Universal Robots PolyScope program: fill_sugar.urp

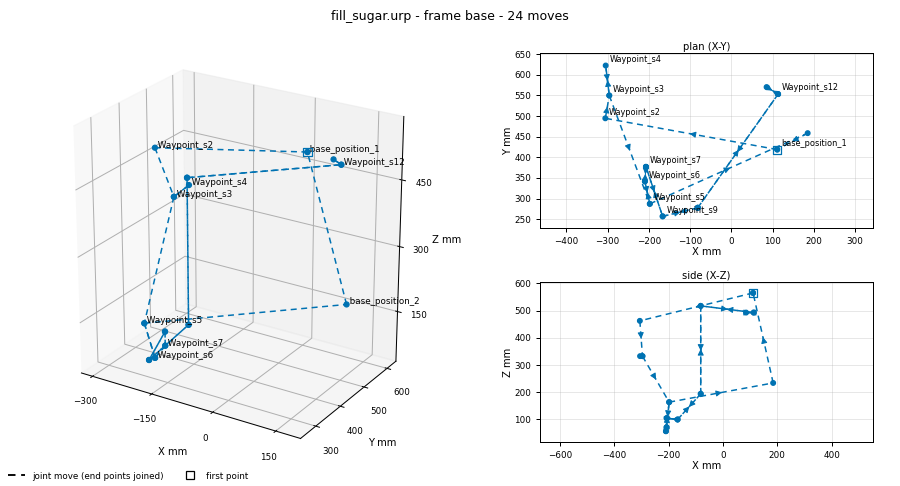
[picture p0: tool path of fill_sugar.urp in frame base, 24 of 24 moves have a stored position in this frame; points joined in program order, loops and branches not executed]
Program fill_sugar (installation=default directory=/programs/Nicolas_Arteaga createdIn=5.12.4.1101661 lastSavedIn=5.12.4.1101661 robotSerialNumber=20225502378)
Calibrated DH parameters: a=[0.00022, -0.425328, -0.389701, 0.000059, 0.000065, 0]; d=[0.162608, 0.803456, 9.992211, -10.662202, 0.099702, 0.099559]; alpha=[1.570756, 0.001543, 0.004316, 1.570651, -1.570122, 0]; deltaTheta=[0, 0.002917, 0.116094, -0.119008, 0, -0.000001]
Robot Program (runOnlyOnce=true)
  'The Sugar Workflow opens the funnel with the sugar the time needed for the amount, moves the spoon into the center of the machine and comes back'
  MoveJ speed 60 deg/s, acceleration 80 deg/s^2 (useActiveTCP=true) feature=Base
    'Use either the register for CPEE or a local parameter like 0.5'
    sugar_amount := GP_int_in[0]
    SuppressedNode
      sugar_amount := 1.5
    Waypoint base_position_1: TCP in base x=110.873 y=418.875 z=565.206 mm, rx=-1.5602 ry=-0.9891 rz=-1.3624 rad; joints [200.91, -129.117, 99.415, 36.172, 41.428, 90] deg; TCP offset x=0 y=0 z=191.5 mm, rx=0 ry=0 rz=0 rad
    Waypoint Waypoint_s2: TCP in base x=-305.749 y=494.617 z=462.545 mm, rx=-1.1337 ry=-1.2693 rz=-1.1298 rad; joints [300.263, -100.211, 102.502, -1.736, 114.115, 89.999] deg; TCP offset x=0 y=0 z=191.5 mm, rx=0 ry=0 rz=0 rad
    URCap Gripper Activate (Robotiq_Grippers, Robotiq Inc.) dataModel(ResetAndActivateKey=false)
    URCap Gripper (Robotiq_Grippers, Robotiq Inc.) dataModel(position=20.0, force=0.0, speed=0.0, positionInDouble=20.0, forceInDouble=0.0, speedInDouble=0.0, slaveIds=[9], blocking=true)
    Waypoint Waypoint_s3: TCP in base x=-296.164 y=549.885 z=332.617 mm, rx=-1.2863 ry=-1.1731 rz=-1.2824 rad; joints [302.576, -85.481, 108.119, -21.976, 128.323, 90.062] deg
    Waypoint Waypoint_s4: TCP in base x=-304.886 y=622.528 z=332.693 mm, rx=-1.2845 ry=-1.1692 rz=-1.2825 rad; joints [298.729, -77.999, 99.501, -20.953, 124.442, 90.195] deg
    URCap Gripper (Robotiq_Grippers, Robotiq Inc.) dataModel(position=35.0, force=100.0, speed=100.0, positionInDouble=35.0, forceInDouble=100.0, speedInDouble=100.0, slaveIds=[9], blocking=true)
    Script: sleep(sugar_amount)
    URCap Gripper (Robotiq_Grippers, Robotiq Inc.) dataModel(position=0.0, force=100.0, speed=0.0, positionInDouble=0.0, forceInDouble=100.0, speedInDouble=0.0, slaveIds=[9], blocking=true)
    Waypoint Waypoint_s3: TCP in base x=-296.164 y=549.885 z=332.617 mm, rx=-1.2863 ry=-1.1731 rz=-1.2824 rad; joints [302.576, -85.481, 108.119, -21.976, 128.323, 90.062] deg
    Waypoint Waypoint_s5: TCP in base x=-197.91 y=287.3 z=163.432 mm, rx=-1.5535 ry=0.1524 rz=-0.1096 rad; joints [326.967, -91.614, 148.2, -58.357, 156.715, 180] deg; TCP offset x=0 y=0 z=191.5 mm, rx=0 ry=0 rz=0 rad
    URCap Gripper (Robotiq_Grippers, Robotiq Inc.) dataModel(position=50.0, force=100.0, speed=0.0, positionInDouble=50.0, forceInDouble=100.0, speedInDouble=0.0, slaveIds=[9], blocking=true)
    Waypoint Waypoint_s6: TCP in base x=-209.858 y=341.762 z=56.515 mm, rx=-1.5807 ry=0.0548 rz=-0.0662 rad; joints [313.143, -65.937, 152.318, -85.713, 137.744, 180] deg; TCP offset x=0 y=0 z=191.5 mm, rx=0 ry=0 rz=0 rad
    Waypoint Waypoint_s7: TCP in base x=-207.363 y=377.054 z=70.962 mm, rx=-1.5764 ry=0.0343 rz=-0.0374 rad; joints [304.137, -69.797, 152.569, -82.518, 126.942, 179.974] deg; TCP offset x=0 y=0 z=191.5 mm, rx=0 ry=0 rz=0 rad
    URCap Gripper (Robotiq_Grippers, Robotiq Inc.) dataModel(position=100.0, force=100.0, speed=0.0, positionInDouble=100.0, forceInDouble=100.0, speedInDouble=0.0, slaveIds=[9], blocking=true)
    Waypoint Waypoint_s8: TCP in base x=-207.108 y=376.646 z=104.52 mm, rx=-1.5811 ry=0.0321 rz=-0.0396 rad; joints [304.156, -79.665, 151.838, -71.558, 126.955, 180.055] deg
    Waypoint Waypoint_s9: TCP in base x=-166.798 y=256.956 z=99.586 mm, rx=-1.5812 ry=0.0311 rz=-0.0496 rad; joints [323.963, -84.01, 161.527, -76.66, 147.1, 180] deg; TCP offset x=0 y=0 z=191.5 mm, rx=0 ry=0 rz=0 rad
    Waypoint Waypoint_s10: TCP in base x=-81.738 y=277.755 z=193.913 mm, rx=-1.6539 ry=-0.0026 rz=-1.0019 rad; joints [319.07, -96.736, 145.387, -56.678, 176.026, 135] deg; TCP offset x=0 y=0 z=191.5 mm, rx=0 ry=0 rz=0 rad
    Waypoint Waypoint_s11: TCP in base x=-81.724 y=277.748 z=517.554 mm, rx=-1.6566 ry=-0.0181 rz=-1.0161 rad; joints [319.137, -114.467, 104.986, 2.526, 175.909, 135] deg; TCP offset x=0 y=0 z=191.5 mm, rx=0 ry=0 rz=0 rad
    Waypoint Waypoint_s12: TCP in base x=113.097 y=553.265 z=492.993 mm, rx=-1.5561 ry=-0.4924 rz=-0.7353 rad; joints [227.113, -110.707, 105.414, 5.953, 56.661, 135.029] deg; TCP offset x=0 y=0 z=191.5 mm, rx=0 ry=0 rz=0 rad
    Waypoint Waypoint_s13: TCP in base x=85.146 y=570.31 z=492.98 mm, rx=-0.6297 ry=-2.0123 rz=-2.0637 rad; joints [234.679, -108.87, 104.254, 5.245, 64.223, 25.001] deg; TCP offset x=0 y=0 z=191.5 mm, rx=0 ry=0 rz=0 rad
    Waypoint Waypoint_s12: TCP in base x=113.097 y=553.265 z=492.993 mm, rx=-1.5561 ry=-0.4924 rz=-0.7353 rad; joints [227.113, -110.707, 105.414, 5.953, 56.661, 135.029] deg; TCP offset x=0 y=0 z=191.5 mm, rx=0 ry=0 rz=0 rad
    Waypoint Waypoint_s11: TCP in base x=-81.724 y=277.748 z=517.554 mm, rx=-1.6566 ry=-0.0181 rz=-1.0161 rad; joints [319.137, -114.467, 104.986, 2.526, 175.909, 135] deg; TCP offset x=0 y=0 z=191.5 mm, rx=0 ry=0 rz=0 rad
    Waypoint Waypoint_s10: TCP in base x=-81.738 y=277.755 z=193.913 mm, rx=-1.6539 ry=-0.0026 rz=-1.0019 rad; joints [319.07, -96.736, 145.387, -56.678, 176.026, 135] deg; TCP offset x=0 y=0 z=191.5 mm, rx=0 ry=0 rz=0 rad
    Waypoint Waypoint_s9: TCP in base x=-166.798 y=256.956 z=99.586 mm, rx=-1.5812 ry=0.0311 rz=-0.0496 rad; joints [323.963, -84.01, 161.527, -76.66, 147.1, 180] deg; TCP offset x=0 y=0 z=191.5 mm, rx=0 ry=0 rz=0 rad
    Waypoint Waypoint_s8: TCP in base x=-207.108 y=376.646 z=104.52 mm, rx=-1.5811 ry=0.0321 rz=-0.0396 rad; joints [304.156, -79.665, 151.838, -71.558, 126.955, 180.055] deg; TCP offset x=0 y=0 z=191.5 mm, rx=0 ry=0 rz=0 rad
    Waypoint Waypoint_s7: TCP in base x=-207.363 y=377.054 z=70.962 mm, rx=-1.5764 ry=0.0343 rz=-0.0374 rad; joints [304.137, -69.797, 152.569, -82.518, 126.942, 179.974] deg
    URCap Gripper (Robotiq_Grippers, Robotiq Inc.) dataModel(position=0.0, force=0.0, speed=100.0, positionInDouble=0.0, forceInDouble=0.0, speedInDouble=100.0, slaveIds=[9], blocking=true)
    Waypoint Waypoint_s6: TCP in base x=-209.858 y=341.762 z=56.515 mm, rx=-1.5807 ry=0.0548 rz=-0.0662 rad; joints [313.143, -65.937, 152.318, -85.713, 137.744, 180] deg; TCP offset x=0 y=0 z=191.5 mm, rx=0 ry=0 rz=0 rad
    Waypoint Waypoint_s5: TCP in base x=-197.91 y=287.3 z=163.432 mm, rx=-1.5535 ry=0.1524 rz=-0.1096 rad; joints [326.967, -91.614, 148.2, -58.357, 156.715, 180] deg; TCP offset x=0 y=0 z=191.5 mm, rx=0 ry=0 rz=0 rad
    Waypoint base_position_2: TCP in base x=184.715 y=458.614 z=234.006 mm, rx=-1.6866 ry=-0.757 rz=-1.7388 rad; joints [237.954, -104.402, 143.977, -41.546, 99.477, 90] deg; TCP offset x=0 y=0 z=191.5 mm, rx=0 ry=0 rz=0 rad
    Waypoint base_position_1: TCP in base x=110.873 y=418.875 z=565.206 mm, rx=-1.5602 ry=-0.9891 rz=-1.3624 rad; joints [200.91, -129.117, 99.415, 36.172, 41.428, 90] deg; TCP offset x=0 y=0 z=191.5 mm, rx=0 ry=0 rz=0 rad
